// TIA Portal V15.1 export
// export: Created 2024-05-17T05:38:40.1335879Z, ExportSetting WithDefaults, DisplayName Totally Integrated Automation Portal, DisplayVersion V15.1 Update 5, DisplayName TIA Portal Openness, DisplayVersion V15.1 Update 5, DisplayName SINAMICS Startdrive Advanced, DisplayVersion V15.1, DisplayName G130, G150, S120, S150, SINAMICS MV, S210, DisplayVersion V15.1, DisplayName G110M, G120, G120C, G120D, G120P, DisplayVersion V15.1, DisplayName STEP 7 Professional, DisplayVersion V15.1 Update 5, DisplayName STEP 7 Safety, DisplayVersion V15.1, DisplayName WinCC Professional, DisplayVersion V15.1 Update 5, DisplayName SIMATIC Visualization Architect, DisplayVersion V15.1
FUNCTION_BLOCK "LGBCrossConvManFnc"   // FB6709, FBD
TITLE = LGBCrossConvManFnc
{ S7_Optimized_Access := 'TRUE' }
VERSION : 0.1
// stored: AutoNumber false, IsIECCheckEnabled false, IsRetainMemResEnabled false, MemoryReserve 100, SetENOAutomatically False, UDAEnableTagReadback false
   VAR_INPUT
      I_LocalPBSet { ExternalAccessible := 'False'; ExternalVisible := 'False'; ExternalWritable := 'False'} : Bool;   // Push button for manual movememt (on local panel) set
      I_LocalPBRes { ExternalAccessible := 'False'; ExternalVisible := 'False'; ExternalWritable := 'False'} : Bool;   // Push button for manual movememt (on local panel) Reset
   END_VAR
   VAR_OUTPUT
      O_ManLSpdSetReq { ExternalAccessible := 'False'; ExternalVisible := 'False'; ExternalWritable := 'False'} : Bool;   // Manual low speed Set request
      O_ManHSpdSetReq { ExternalAccessible := 'False'; ExternalVisible := 'False'; ExternalWritable := 'False'} : Bool;   // Manual high speed Set request
      O_ManLSpdResReq { ExternalAccessible := 'False'; ExternalVisible := 'False'; ExternalWritable := 'False'} : Bool;   // Manual low speed Reset request
      O_ManHSpdResReq { ExternalAccessible := 'False'; ExternalVisible := 'False'; ExternalWritable := 'False'} : Bool;   // Manual high speed Reset request
      O_ManSetReq { ExternalAccessible := 'False'; ExternalVisible := 'False'; ExternalWritable := 'False'} : Bool;   // Manual Set request
      O_ManResReq { ExternalAccessible := 'False'; ExternalVisible := 'False'; ExternalWritable := 'False'} : Bool;   // Manual Res request
   END_VAR
   VAR_IN_OUT
      H_HMICmd { ExternalAccessible := 'False'; ExternalVisible := 'False'; ExternalWritable := 'False'} : Word;   // HMI Command
      H_HMICmdOnScreenAsNext { ExternalAccessible := 'False'; ExternalVisible := 'False'; ExternalWritable := 'False'} : Word;   // HMI Command on HMI screen as Next / HMI Command
      H_HMICmdOnScreenAsPrev { ExternalAccessible := 'False'; ExternalVisible := 'False'; ExternalWritable := 'False'} : Word;   // HMI Command on HMI screen as Previous / HMI Command
      IO_Modes : "Modes";   // Modes
      IO_ModesOnScreenAsNext : "Modes";   // Modes / Modes on HMI screen as Next
      IO_ModesOnScreenAsPrev : "Modes";   // Modes / Modes on HMI screen as Previous
      H_HMI : "H_HMI";   // HMI Command
      H_HMIPrevCC : "H_HMI";   // HMI Command Previous / HMI Command
      H_HMINextCC : "H_HMI";   // HMI Command Next / HMI Command
   END_VAR
   VAR
      ManLSpdSetReq { ExternalAccessible := 'False'; ExternalVisible := 'False'; ExternalWritable := 'False'} : Bool;   // Manual low speed Set request
      ManHSpdSetReq { ExternalAccessible := 'False'; ExternalVisible := 'False'; ExternalWritable := 'False'} : Bool;   // Manual high speed Set request
      ManLSpdResReq { ExternalAccessible := 'False'; ExternalVisible := 'False'; ExternalWritable := 'False'} : Bool;   // Manual low speed Reset request
      ManHSpdResReq { ExternalAccessible := 'False'; ExternalVisible := 'False'; ExternalWritable := 'False'} : Bool;   // Manual high speed Reset request
      Edge { ExternalAccessible := 'False'; ExternalVisible := 'False'; ExternalWritable := 'False'} : Array[1..10] of Bool;   // Edge
      PulsFncSel { ExternalAccessible := 'False'; ExternalVisible := 'False'; ExternalWritable := 'False'} : TP_TIME;   // Timer
   END_VAR
   VAR_TEMP
      H_CommandDW1 : Struct
         SelectOnAnotherScreen : Bool;
         SelectAsNext : Bool;
         SelectAsPrevious : Bool;
         Bit3 : Bool;
         Bit4 : Bool;
         Bit5 : Bool;
         Bit6 : Bool;
         Bit7 : Bool;
         Bit8 : Bool;
         Bit9 : Bool;
         Bit10 : Bool;
         Bit11 : Bool;
         Bit12 : Bool;
         Bit13 : Bool;
         Bit14 : Bool;
         Bit15 : Bool;
         Bit16 : Bool;
         Bit17 : Bool;
         Bit18 : Bool;
         Bit19 : Bool;
         Bit20 : Bool;
         Bit21 : Bool;
         Bit22 : Bool;
         Bit23 : Bool;
         Bit24 : Bool;
         Bit25 : Bool;
         Bit26 : Bool;
         Bit27 : Bool;
         Bit28 : Bool;
         Bit29 : Bool;
         Bit30 : Bool;
         Bit31 : Bool;
      END_STRUCT;
   END_VAR
   VAR_TEMP   // added for the SCL form of the ladder/FBD networks
      _w1 : Bool;
      _w2 : Bool;
      _w3 : Bool;
      _w4 : Bool;
      _w5 : Bool;
   END_VAR
BEGIN

REGION Network 1: **** 1 - Inputs **** Extract HMI Commands
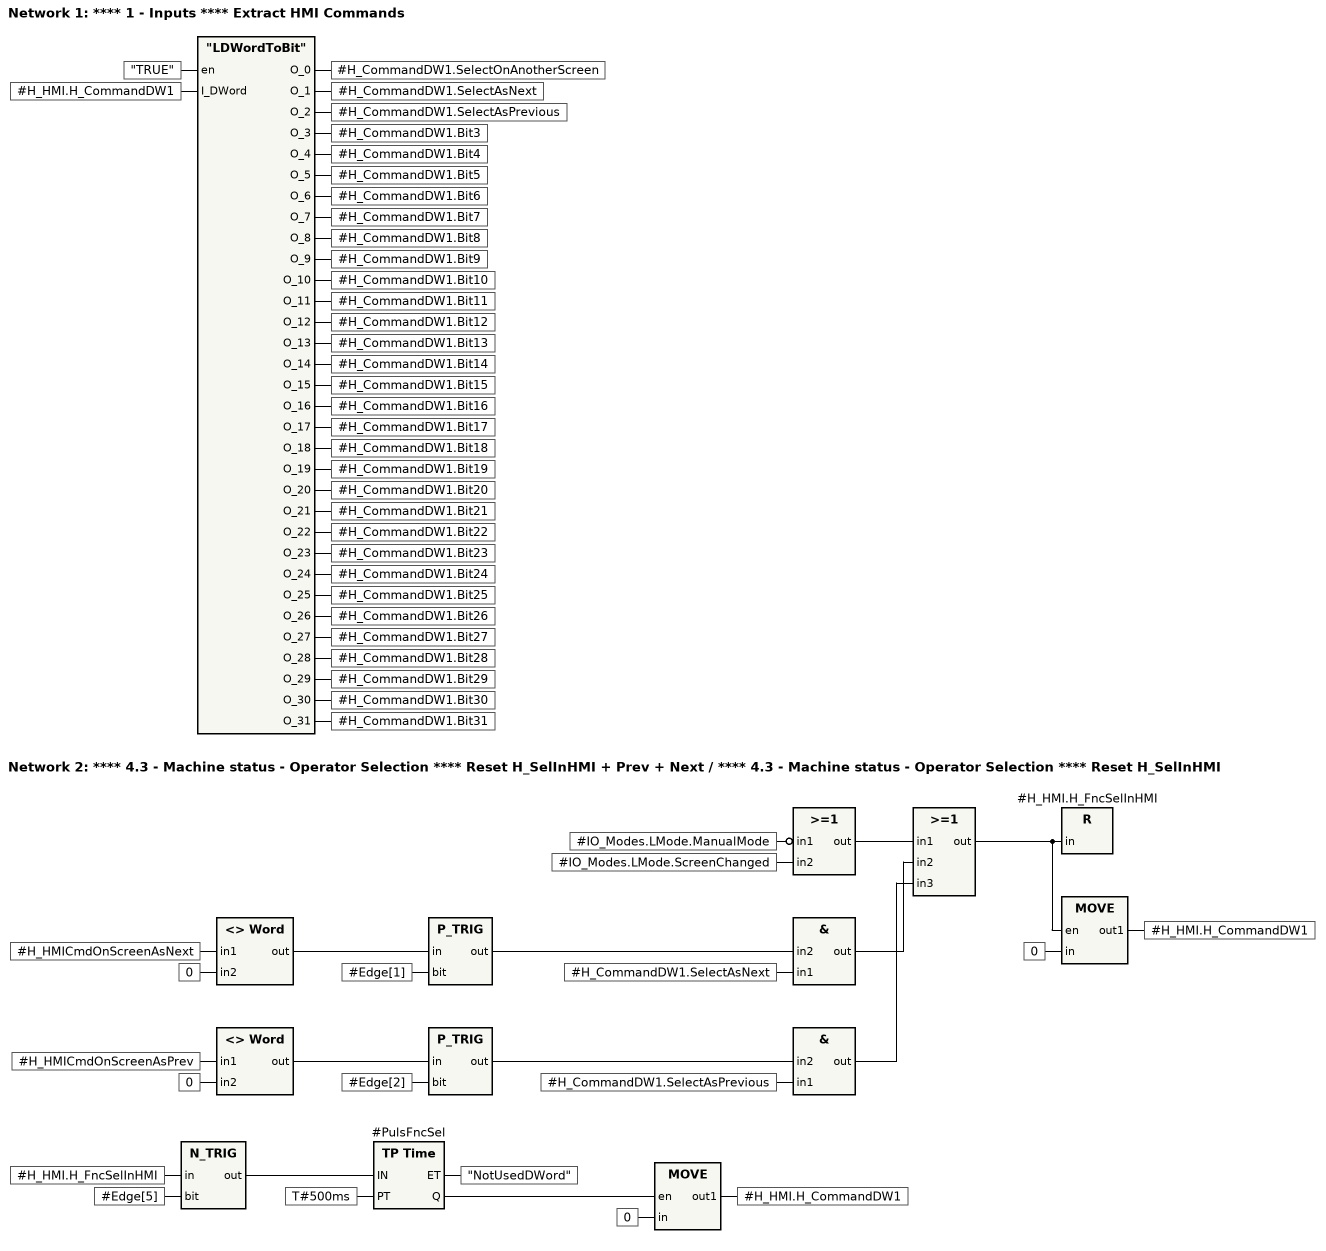
   IF "TRUE" THEN
       "LDWordToBit"(I_DWord := #H_HMI.H_CommandDW1,
                     O_0 => #H_CommandDW1.SelectOnAnotherScreen,
                     O_1 => #H_CommandDW1.SelectAsNext,
                     O_2 => #H_CommandDW1.SelectAsPrevious,
                     O_3 => #H_CommandDW1.Bit3,
                     O_4 => #H_CommandDW1.Bit4,
                     O_5 => #H_CommandDW1.Bit5,
                     O_6 => #H_CommandDW1.Bit6,
                     O_7 => #H_CommandDW1.Bit7,
                     O_8 => #H_CommandDW1.Bit8,
                     O_9 => #H_CommandDW1.Bit9,
                     O_10 => #H_CommandDW1.Bit10,
                     O_11 => #H_CommandDW1.Bit11,
                     O_12 => #H_CommandDW1.Bit12,
                     O_13 => #H_CommandDW1.Bit13,
                     O_14 => #H_CommandDW1.Bit14,
                     O_15 => #H_CommandDW1.Bit15,
                     O_16 => #H_CommandDW1.Bit16,
                     O_17 => #H_CommandDW1.Bit17,
                     O_18 => #H_CommandDW1.Bit18,
                     O_19 => #H_CommandDW1.Bit19,
                     O_20 => #H_CommandDW1.Bit20,
                     O_21 => #H_CommandDW1.Bit21,
                     O_22 => #H_CommandDW1.Bit22,
                     O_23 => #H_CommandDW1.Bit23,
                     O_24 => #H_CommandDW1.Bit24,
                     O_25 => #H_CommandDW1.Bit25,
                     O_26 => #H_CommandDW1.Bit26,
                     O_27 => #H_CommandDW1.Bit27,
                     O_28 => #H_CommandDW1.Bit28,
                     O_29 => #H_CommandDW1.Bit29,
                     O_30 => #H_CommandDW1.Bit30,
                     O_31 => #H_CommandDW1.Bit31);
   END_IF;
END_REGION

REGION Network 2: **** 4.3 - Machine status - Operator Selection **** Reset H_SelInHMI + Prev + Next / **** 4.3 - Machine status - Operator Selection **** Reset H_SelInHMI
   #_w1 := #H_HMICmdOnScreenAsNext <> 0;
   #_w2 := #_w1 AND NOT #Edge[1];   // rising edge
   #Edge[1] := #_w1;
   #_w3 := #H_HMICmdOnScreenAsPrev <> 0;
   #_w4 := #_w3 AND NOT #Edge[2];   // rising edge
   #Edge[2] := #_w3;
   IF NOT #IO_Modes.LMode.ManualMode OR #IO_Modes.LMode.ScreenChanged OR (#_w2 AND #H_CommandDW1.SelectAsNext) OR (#_w4 AND #H_CommandDW1.SelectAsPrevious) THEN
       #H_HMI.H_FncSelInHMI := FALSE;
       #H_HMI.H_CommandDW1 := 0;
   END_IF;
   #_w5 := NOT #H_HMI.H_FncSelInHMI AND #Edge[5];   // falling edge
   #Edge[5] := #H_HMI.H_FncSelInHMI;
   #PulsFncSel(IN := #_w5, PT := T#500ms, ET => "NotUsedDWord");   // TP
   IF #PulsFncSel.Q THEN #H_HMI.H_CommandDW1 := 0; END_IF;
END_REGION

REGION Network 3: **** 4.3 - Machine status - Operator Selection **** Reset HMI Commands
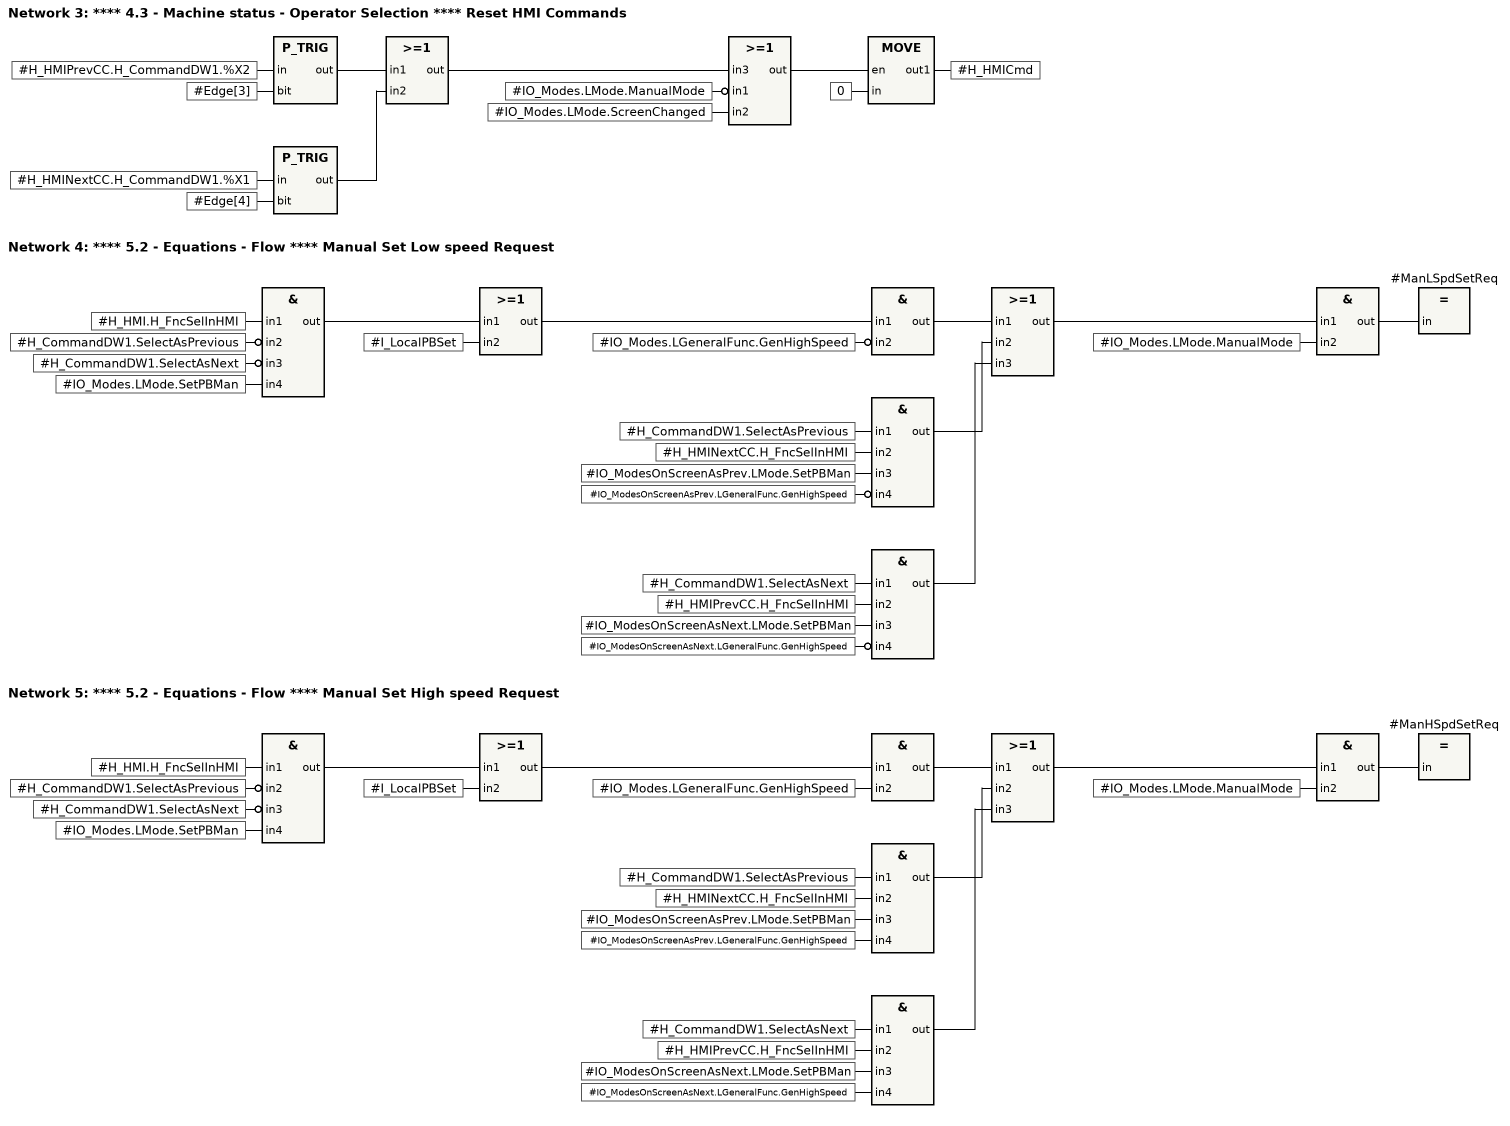
   #_w1 := #H_HMIPrevCC.H_CommandDW1.%X2 AND NOT #Edge[3];   // rising edge
   #Edge[3] := #H_HMIPrevCC.H_CommandDW1.%X2;
   #_w2 := #H_HMINextCC.H_CommandDW1.%X1 AND NOT #Edge[4];   // rising edge
   #Edge[4] := #H_HMINextCC.H_CommandDW1.%X1;
   IF #_w1 OR #_w2 OR NOT #IO_Modes.LMode.ManualMode OR #IO_Modes.LMode.ScreenChanged THEN
       #H_HMICmd := 0;
   END_IF;
END_REGION

REGION Network 4: **** 5.2 - Equations - Flow **** Manual Set Low speed Request
   #ManLSpdSetReq := ((((#H_HMI.H_FncSelInHMI AND NOT #H_CommandDW1.SelectAsPrevious AND NOT #H_CommandDW1.SelectAsNext AND #IO_Modes.LMode.SetPBMan) OR #I_LocalPBSet) AND NOT #IO_Modes.LGeneralFunc.GenHighSpeed) OR (#H_CommandDW1.SelectAsPrevious AND #H_HMINextCC.H_FncSelInHMI AND #IO_ModesOnScreenAsPrev.LMode.SetPBMan AND NOT #IO_ModesOnScreenAsPrev.LGeneralFunc.GenHighSpeed) OR (#H_CommandDW1.SelectAsNext AND #H_HMIPrevCC.H_FncSelInHMI AND #IO_ModesOnScreenAsNext.LMode.SetPBMan AND NOT #IO_ModesOnScreenAsNext.LGeneralFunc.GenHighSpeed)) AND #IO_Modes.LMode.ManualMode;
END_REGION

REGION Network 5: **** 5.2 - Equations - Flow **** Manual Set High speed Request
   #ManHSpdSetReq := ((((#H_HMI.H_FncSelInHMI AND NOT #H_CommandDW1.SelectAsPrevious AND NOT #H_CommandDW1.SelectAsNext AND #IO_Modes.LMode.SetPBMan) OR #I_LocalPBSet) AND #IO_Modes.LGeneralFunc.GenHighSpeed) OR (#H_CommandDW1.SelectAsPrevious AND #H_HMINextCC.H_FncSelInHMI AND #IO_ModesOnScreenAsPrev.LMode.SetPBMan AND #IO_ModesOnScreenAsPrev.LGeneralFunc.GenHighSpeed) OR (#H_CommandDW1.SelectAsNext AND #H_HMIPrevCC.H_FncSelInHMI AND #IO_ModesOnScreenAsNext.LMode.SetPBMan AND #IO_ModesOnScreenAsNext.LGeneralFunc.GenHighSpeed)) AND #IO_Modes.LMode.ManualMode;
END_REGION

REGION Network 6: **** 5.2 - Equations - Flow **** Manual Reset Low speed Request
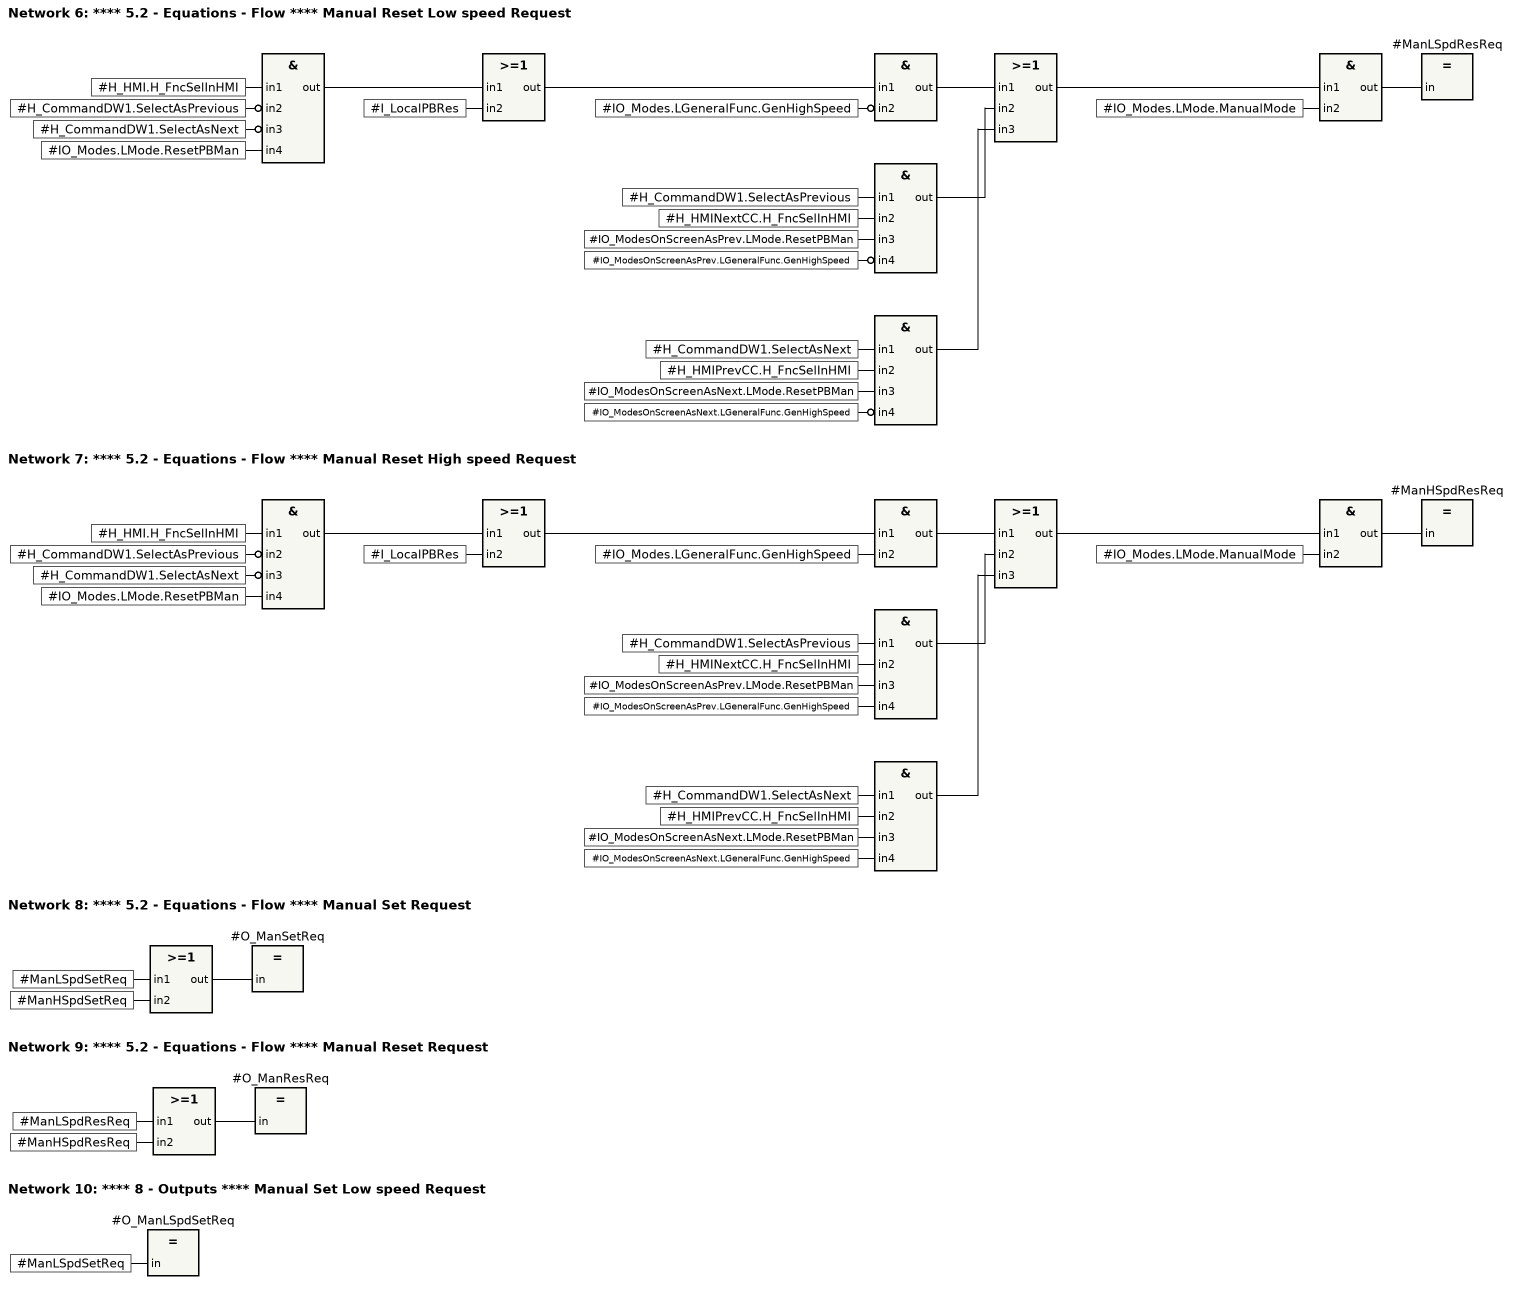
   #ManLSpdResReq := ((((#H_HMI.H_FncSelInHMI AND NOT #H_CommandDW1.SelectAsPrevious AND NOT #H_CommandDW1.SelectAsNext AND #IO_Modes.LMode.ResetPBMan) OR #I_LocalPBRes) AND NOT #IO_Modes.LGeneralFunc.GenHighSpeed) OR (#H_CommandDW1.SelectAsPrevious AND #H_HMINextCC.H_FncSelInHMI AND #IO_ModesOnScreenAsPrev.LMode.ResetPBMan AND NOT #IO_ModesOnScreenAsPrev.LGeneralFunc.GenHighSpeed) OR (#H_CommandDW1.SelectAsNext AND #H_HMIPrevCC.H_FncSelInHMI AND #IO_ModesOnScreenAsNext.LMode.ResetPBMan AND NOT #IO_ModesOnScreenAsNext.LGeneralFunc.GenHighSpeed)) AND #IO_Modes.LMode.ManualMode;
END_REGION

REGION Network 7: **** 5.2 - Equations - Flow **** Manual Reset High speed Request
   #ManHSpdResReq := ((((#H_HMI.H_FncSelInHMI AND NOT #H_CommandDW1.SelectAsPrevious AND NOT #H_CommandDW1.SelectAsNext AND #IO_Modes.LMode.ResetPBMan) OR #I_LocalPBRes) AND #IO_Modes.LGeneralFunc.GenHighSpeed) OR (#H_CommandDW1.SelectAsPrevious AND #H_HMINextCC.H_FncSelInHMI AND #IO_ModesOnScreenAsPrev.LMode.ResetPBMan AND #IO_ModesOnScreenAsPrev.LGeneralFunc.GenHighSpeed) OR (#H_CommandDW1.SelectAsNext AND #H_HMIPrevCC.H_FncSelInHMI AND #IO_ModesOnScreenAsNext.LMode.ResetPBMan AND #IO_ModesOnScreenAsNext.LGeneralFunc.GenHighSpeed)) AND #IO_Modes.LMode.ManualMode;
END_REGION

REGION Network 8: **** 5.2 - Equations - Flow **** Manual Set Request
   #O_ManSetReq := #ManLSpdSetReq OR #ManHSpdSetReq;
END_REGION

REGION Network 9: **** 5.2 - Equations - Flow **** Manual Reset Request
   #O_ManResReq := #ManLSpdResReq OR #ManHSpdResReq;
END_REGION

REGION Network 10: **** 8 - Outputs **** Manual Set Low speed Request
   #O_ManLSpdSetReq := #ManLSpdSetReq;
END_REGION

REGION Network 11: **** 8 - Outputs **** Manual high speed Set request
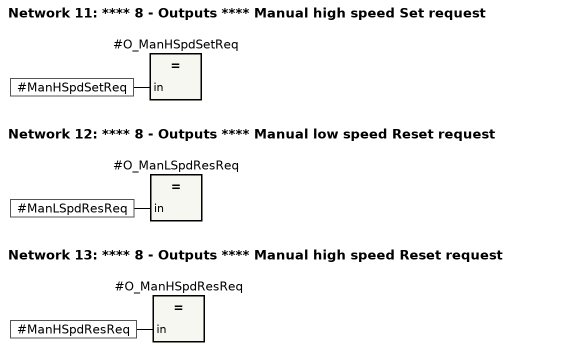
   #O_ManHSpdSetReq := #ManHSpdSetReq;
END_REGION

REGION Network 12: **** 8 - Outputs **** Manual low speed Reset request
   #O_ManLSpdResReq := #ManLSpdResReq;
END_REGION

REGION Network 13: **** 8 - Outputs **** Manual high speed Reset request
   #O_ManHSpdResReq := #ManHSpdResReq;
END_REGION
END_FUNCTION_BLOCK
